KUKA KRL program: ho_lca_st03_pos03.src, ho_lca_st03_pos03.dat

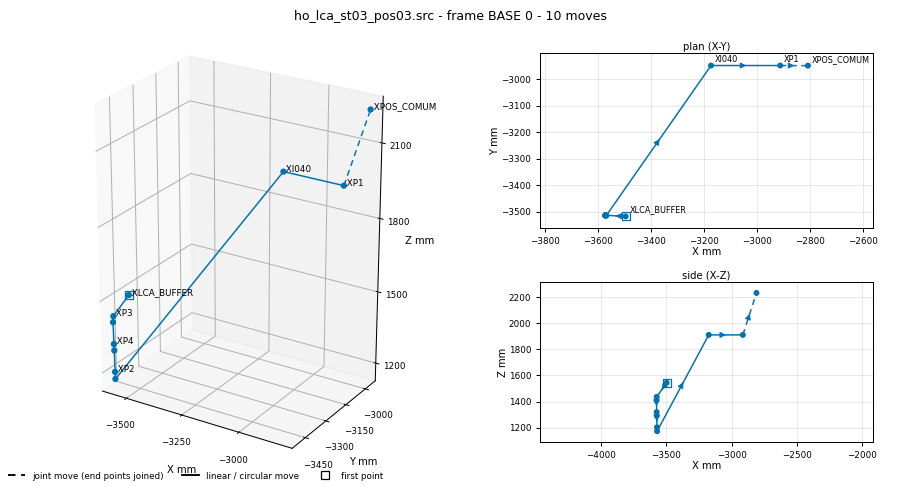
[picture p0: tool path of ho_lca_st03_pos03.src in frame BASE 0, 10 of 10 moves have a stored position in this frame; points joined in program order, loops and branches not executed]
--- ho_lca_st03_pos03.src ---
&ACCESS RVO4
&REL 18
&COMMENT POS_3 LCA
&PARAM DISKPATH = KRC:\R1\Program\LCA
&PARAM TEMPLATE = C:\KRC\Roboter\Template\vorgabe
&PARAM EDITMASK = *
DEF ho_lca_st03_pos03( )
;FOLD INI
  ;FOLD BASISTECH INI
    GLOBAL INTERRUPT DECL 3 WHEN $STOPMESS==TRUE DO IR_STOPM ( )
    INTERRUPT ON 3
    BAS (#INITMOV,0 )
  ;ENDFOLD (BASISTECH INI)
;FOLD GRIPPERTECH INI
USER_GRP(0,DUMMY,DUMMY,GDEFAULT)
;ENDFOLD (GRIPPERTECH INI)
  ;FOLD USER INI
    ;Make your modifications here

  ;ENDFOLD (USER INI)
;ENDFOLD (INI)

; Caracterizacao dos meios de producao:
; Changes: Pega LCA Posicao 3 (Pc-3)
; Versao Atual: 14/08/2015
; Name: P13.050-R2

;FOLD PTP LCA_BUFFER Vel=100 % DEFAULT Tool[15]:AUX_LCA Base[0];%{PE}%R 8.2.20,%MKUKATPBASIS,%CMOVE,%VPTP,%P 1:PTP, 2:LCA_BUFFER, 3:, 5:100, 7:DEFAULT
$BWDSTART=FALSE
PDAT_ACT=PDEFAULT
FDAT_ACT=FLCA_BUFFER
BAS(#PTP_PARAMS,100)
PTP XLCA_BUFFER
;ENDFOLD

;FOLD WAIT FOR ( IN 3362 'LCA p.3' );%{PE}%R 8.2.20,%MKUKATPBASIS,%CEXT_WAIT_FOR,%VEXT_WAIT_FOR,%P 2:, 4:, 5:$IN, 6:3362, 7:LCA p.3, 9:
WAIT FOR  ( $IN[3362] )
;ENDFOLD

;FOLD LIN P3 Vel=1 m/s CPDAT3 Tool[15]:AUX_LCA Base[0];%{PE}%R 8.2.20,%MKUKATPBASIS,%CMOVE,%VLIN,%P 1:LIN, 2:P3, 3:, 5:1, 7:CPDAT3
$BWDSTART=FALSE
LDAT_ACT=LCPDAT3
FDAT_ACT=FP3
BAS(#CP_PARAMS,1)
LIN XP3
;ENDFOLD

;FOLD WAIT FOR ( NOT IN 489 'Presença de peça 1 - Axor LCA' );%{PE}%R 8.2.20,%MKUKATPBASIS,%CEXT_WAIT_FOR,%VEXT_WAIT_FOR,%P 2:, 4:NOT, 5:$IN, 6:489, 7:Presença de peça 1 - Axor LCA, 9:
WAIT FOR  (  NOT $IN[489] )
;ENDFOLD

;FOLD ; POSIÇÃO 1 LCA AUSENTE;%{PE}%R 8.2.20,%MKUKATPBASIS,%CCOMMENT,%VNORMAL,%P 2:POSIÇÃO 1 LCA  AUSENTE
;ENDFOLD
;FOLD LIN PEGA_1 Vel=0.05 m/s L_OLP7 Tool[15]:AUX_LCA Base[0];%{PE}%R 8.2.20,%MKUKATPBASIS,%CMOVE,%VLIN,%P 1:LIN, 2:PEGA_1, 3:, 5:0.05, 7:L_OLP7
$BWDSTART=FALSE
LDAT_ACT=LL_OLP7
FDAT_ACT=FPEGA_1
BAS(#CP_PARAMS,0.05)
LIN XPEGA_1
;ENDFOLD

;FOLD LIN P4 Vel=0.05 m/s CPDAT4 Tool[15]:AUX_LCA Base[0];%{PE}%R 8.2.20,%MKUKATPBASIS,%CMOVE,%VLIN,%P 1:LIN, 2:P4, 3:, 5:0.05, 7:CPDAT4
$BWDSTART=FALSE
LDAT_ACT=LCPDAT4
FDAT_ACT=FP4
BAS(#CP_PARAMS,0.05)
LIN XP4
;ENDFOLD

;FOLD WAIT FOR ( NOT IN 489 'Presença de peça 1 - Axor LCA' );%{PE}%R 8.2.20,%MKUKATPBASIS,%CEXT_WAIT_FOR,%VEXT_WAIT_FOR,%P 2:, 4:NOT, 5:$IN, 6:489, 7:Presença de peça 1 - Axor LCA, 9:
WAIT FOR  (  NOT $IN[489] )
;ENDFOLD

;FOLD ; POSIÇÃO 2 LCA AUSENTE;%{PE}%R 8.2.20,%MKUKATPBASIS,%CCOMMENT,%VNORMAL,%P 2:POSIÇÃO 2 LCA  AUSENTE
;ENDFOLD
;FOLD LIN PEGA_2 Vel=0.05 m/s L_OLP8 Tool[15]:AUX_LCA Base[0];%{PE}%R 8.2.20,%MKUKATPBASIS,%CMOVE,%VLIN,%P 1:LIN, 2:PEGA_2, 3:, 5:0.05, 7:L_OLP8
$BWDSTART=FALSE
LDAT_ACT=LL_OLP8
FDAT_ACT=FPEGA_2
BAS(#CP_PARAMS,0.05)
LIN XPEGA_2
;ENDFOLD

;FOLD LIN P2 Vel=0.05 m/s CPDAT2 Tool[15]:AUX_LCA Base[0];%{PE}%R 8.2.20,%MKUKATPBASIS,%CMOVE,%VLIN,%P 1:LIN, 2:P2, 3:, 5:0.05, 7:CPDAT2
$BWDSTART=FALSE
LDAT_ACT=LCPDAT2
FDAT_ACT=FP2
BAS(#CP_PARAMS,0.05)
LIN XP2
;ENDFOLD

;FOLD ; POSIÇÃO 3 DE PEGA DA PEÇA;%{PE}%R 8.2.20,%MKUKATPBASIS,%CCOMMENT,%VNORMAL,%P 2:POSIÇÃO  3 DE PEGA DA PEÇA
;ENDFOLD
;FOLD LIN PEGA_3 Vel=0.05 m/s L_OLP5 Tool[15]:AUX_LCA Base[0];%{PE}%R 8.2.20,%MKUKATPBASIS,%CMOVE,%VLIN,%P 1:LIN, 2:PEGA_3, 3:, 5:0.05, 7:L_OLP5
$BWDSTART=FALSE
LDAT_ACT=LL_OLP5
FDAT_ACT=FPEGA_3
BAS(#CP_PARAMS,0.05)
LIN XPEGA_3
;ENDFOLD

IF (NOT(GHOST())) THEN
;FOLD WAIT FOR ( IN 489 'Presença de peça 1 - Axor' );%{PE}%R 8.2.20,%MKUKATPBASIS,%CEXT_WAIT_FOR,%VEXT_WAIT_FOR,%P 2:, 4:, 5:$IN, 6:489, 7:Presença de peça 1 - Axor, 9:
WAIT FOR  ( $IN[489] )
;ENDFOLD
ENDIF

;FOLD SET Z4.1 GRP AXOR State=CLO GDAT6;%{PE}%R 8.2.1,%MKUKATPGRP,%CGRP,%VGRP,%P 2:12, 4:2, 5:#NO, 6:GDAT6, 8:0, 10:0
H50(GRP,12,2,GGDAT6)
;ENDFOLD
chk_w6_grp4_clo()

IF (NOT(GHOST())) THEN
;FOLD SET VACUO AXOR State=VACUUM GDAT7;%{PE}%R 8.2.1,%MKUKATPGRP,%CGRP,%VGRP,%P 2:9, 4:1, 5:#NO, 6:GDAT7, 8:0, 10:0
H50(GRP,9,1,GGDAT7)
;ENDFOLD
chk_w6_grp1_vac()
ENDIF

;FOLD OUT 3371 'Lib. p/ sair c/ Travessa Axor/Atego' State=TRUE ;%{PE}%R 8.2.20,%MKUKATPBASIS,%COUT,%VOUTX,%P 2:3371, 3:Lib. p/ sair c/ Travessa Axor/Atego, 5:TRUE, 6:
$OUT[3371]=TRUE
;ENDFOLD
;FOLD WAIT Time=1 sec;%{PE}%R 8.2.20,%MKUKATPBASIS,%CWAIT,%VWAIT,%P 3:1
WAIT SEC 1
;ENDFOLD
;FOLD WAIT FOR ( IN 3371 'Lib. p/ Sair c/ Pç LCA Axor/Atego' );%{PE}%R 8.2.20,%MKUKATPBASIS,%CEXT_WAIT_FOR,%VEXT_WAIT_FOR,%P 2:, 4:, 5:$IN, 6:3371, 7:Lib. p/ Sair c/ Pç LCA Axor/Atego, 9:
WAIT FOR  ( $IN[3371] )
;ENDFOLD
;FOLD OUT 3371 'Lib. p/ sair c/ Travessa Axor/Atego' State=FALSE ;%{PE}%R 8.2.20,%MKUKATPBASIS,%COUT,%VOUTX,%P 2:3371, 3:Lib. p/ sair c/ Travessa Axor/Atego, 5:FALSE, 6:
$OUT[3371]=FALSE
;ENDFOLD
;FOLD OUT 3349 'R2 pegou peça' State=FALSE ;%{PE}%R 8.2.20,%MKUKATPBASIS,%COUT,%VOUTX,%P 2:3349, 3:R2 pegou peça, 5:FALSE, 6:
$OUT[3349]=FALSE
;ENDFOLD

;FOLD LIN l040 Vel=0.02 m/s L_OLP6 Tool[6]:Gripper G0100R Base[0];%{PE}%R 8.2.20,%MKUKATPBASIS,%CMOVE,%VLIN,%P 1:LIN, 2:l040, 3:, 5:0.02, 7:L_OLP6
$BWDSTART=FALSE
LDAT_ACT=LL_OLP6
FDAT_ACT=Fl040
BAS(#CP_PARAMS,0.02)
LIN Xl040
;ENDFOLD

;FOLD WAIT FOR ( IN 489 'Presença de peça 1 - Axor LCA' OR Ghost() );%{PE}%R 8.2.20,%MKUKATPBASIS,%CEXT_WAIT_FOR,%VEXT_WAIT_FOR,%P 2:, 4:, 5:$IN, 6:489, 7:Presença de peça 1 - Axor LCA, 8:OR, 9:, 10:Ghost(), 11:489, 12:, 14:
WAIT FOR  ( $IN[489] OR Ghost() )
;ENDFOLD

;FOLD LIN P1 Vel=0.05 m/s CPDAT1 Tool[6]:Gripper G0100R Base[0];%{PE}%R 8.2.20,%MKUKATPBASIS,%CMOVE,%VLIN,%P 1:LIN, 2:P1, 3:, 5:0.05, 7:CPDAT1
$BWDSTART=FALSE
LDAT_ACT=LCPDAT1
FDAT_ACT=FP1
BAS(#CP_PARAMS,0.05)
LIN XP1
;ENDFOLD

;FOLD ; POSIÇÃO COMUM;%{PE}%R 8.2.20,%MKUKATPBASIS,%CCOMMENT,%VNORMAL,%P 2:POSIÇÃO COMUM
;ENDFOLD
;FOLD PTP POS_COMUM Vel=100 % PDAT0 Tool[6]:Gripper G0100R Base[0];%{PE}%R 8.2.20,%MKUKATPBASIS,%CMOVE,%VPTP,%P 1:PTP, 2:POS_COMUM, 3:, 5:100, 7:PDAT0
$BWDSTART=FALSE
PDAT_ACT=PPDAT0
FDAT_ACT=FPOS_COMUM
BAS(#PTP_PARAMS,100)
PTP XPOS_COMUM
;ENDFOLD

END

--- ho_lca_st03_pos03.dat ---
&ACCESS RVO4
&REL 18
&COMMENT POS_3 LCA
&PARAM DISKPATH = KRC:\R1\Program\LCA
&PARAM TEMPLATE = C:\KRC\Roboter\Template\vorgabe
&PARAM EDITMASK = *
DEFDAT  ho_lca_st03_pos03
;FOLD EXTERNAL DECLARATIONS;%{PE}%MKUKATPBASIS,%CEXT,%VCOMMON,%P
;FOLD GRIPPERTECH EXT
EXT  H50 (INT  :IN,INT  :IN,INT  :IN,GRP_TYP  :IN )
;ENDFOLD (GRIPPERTECH EXT)
;FOLD SPOTTECH EXT
EXT  USERSPOT (S_COMMAND  :IN,SPOT_TYPE  :IN )
;ENDFOLD (SPOTTECH EXT)
;FOLD BASISTECH EXT;%{PE}%MKUKATPBASIS,%CEXT,%VEXT,%P
EXT  BAS (BAS_COMMAND  :IN,REAL  :IN )
DECL INT SUCCESS
;ENDFOLD (BASISTECH EXT)
;FOLD USER EXT;%{E}%MKUKATPUSER,%CEXT,%VEXT,%P
;Make your modifications here

;ENDFOLD (USER EXT)
;ENDFOLD (EXTERNAL DECLARATIONS)
DECL BASIS_SUGG_T LAST_BASIS={POINT1[] "P4                      ",POINT2[] "P4                      ",CP_PARAMS[] "CPDAT4                  ",PTP_PARAMS[] "PDAT0                   ",CONT[] "                        ",CP_VEL[] "0.05                    ",PTP_VEL[] "100                     ",SYNC_PARAMS[] "SYNCDAT                 ",SPL_NAME[] "S0                      "}
DECL LDAT LL_OLP5={VEL 0.25,ACC 100.0,APO_DIST 0.0,APO_FAC 0.0,ORI_TYP #VAR,CIRC_TYP #BASE,JERK_FAC 50.0}
DECL GRP_SUGG_T LAST_GRP={NUMBER[] "9                       ",STATE[] "1                       ",PARAMS[] "GDAT1                   "}
DECL GRP_TYP GGDAT6={G_APO #NO,GRP_TIME 0.200000003,CTRL #OFF,DLY 0,DST 1}
DECL LDAT LL_OLP6={VEL 0.25,ACC 100.0,APO_DIST 0.0,APO_FAC 0.0,ORI_TYP #VAR,CIRC_TYP #BASE,JERK_FAC 50.0}
DECL E6POS Xl040={X -3174.60205,Y -2948.20093,Z 1910.30298,A -158.906006,B 84.1113815,C 96.0123901,S 2,T 34,E1 3299.98706,E2 0.0,E3 0.0,E4 0.0,E5 0.0,E6 0.0}
DECL FDAT Fl040={TOOL_NO 6,BASE_NO 0,IPO_FRAME #BASE,POINT2[] " ",TQ_STATE FALSE}
DECL GRP_TYP GGDAT1={G_APO #NO,GRP_TIME 0.200000003,CTRL #OFF,DLY 0,DST 1}
DECL GRP_TYP GGDAT2={G_APO #NO,GRP_TIME 0.200000003,CTRL #OFF,DLY 0,DST 1}
DECL PDAT PPDAT0={VEL 100.0,ACC 100.0,APO_DIST 100.0}
DECL E6POS XPOS_COMUM={X -2809.396,Y -2948.65088,Z 2231.30811,A -163.868805,B 82.3905334,C 90.4837494,S 2,T 34,E1 3299.98706,E2 0.0,E3 0.0,E4 0.0,E5 0.0,E6 0.0}
DECL FDAT FPOS_COMUM={TOOL_NO 6,BASE_NO 0,IPO_FRAME #BASE,POINT2[] " ",TQ_STATE FALSE}
DECL GRP_TYP GGDAT3={G_APO #NO,GRP_TIME 0.200000003,CTRL #OFF,DLY 0,DST 1}
DECL GRP_TYP GGDAT4={G_APO #NO,GRP_TIME 0.200000003,CTRL #OFF,DLY 0,DST 1}
DECL E6POS XP1={X -2913.604,Y -2948.19995,Z 1910.297,A -158.903305,B 84.1116409,C 96.0151291,S 2,T 34,E1 3299.98706,E2 0.0,E3 0.0,E4 0.0,E5 0.0,E6 0.0}
DECL FDAT FP1={TOOL_NO 6,BASE_NO 0,IPO_FRAME #BASE,POINT2[] " ",TQ_STATE FALSE}
DECL LDAT LCPDAT1={VEL 2.0,ACC 100.0,APO_DIST 100.0,APO_FAC 50.0,AXIS_VEL 100.0,AXIS_ACC 100.0,ORI_TYP #VAR,CIRC_TYP #BASE,JERK_FAC 50.0,GEAR_JERK 50.0,EXAX_IGN 0}
DECL GRP_TYP GGDAT5={G_APO #NO,GRP_TIME 0.200000003,CTRL #OFF,DLY 0,DST 1}
DECL GRP_TYP GGDAT7={G_APO #NO,GRP_TIME 0.200000003,CTRL #OFF,DLY 0,DST 1}
DECL E6POS XLCA_BUFFER={X -3496.6189,Y -3516.89502,Z 1544.35803,A -172.404495,B -1.92999804,C -179.6474,S 2,T 34,E1 3299.98901,E2 0.0,E3 0.0,E4 0.0,E5 0.0,E6 0.0}
DECL FDAT FLCA_BUFFER={TOOL_NO 15,BASE_NO 0,IPO_FRAME #BASE,POINT2[] " ",TQ_STATE FALSE}
DECL E6POS XP2={X -3570.20801,Y -3514.07397,Z 1203.78003,A -172.936798,B -0.115350299,C 179.957001,S 2,T 34,E1 3299.98511,E2 0.0,E3 0.0,E4 0.0,E5 0.0,E6 0.0}
DECL FDAT FP2={TOOL_NO 15,BASE_NO 0,IPO_FRAME #BASE,POINT2[] " ",TQ_STATE FALSE}
DECL LDAT LCPDAT2={VEL 2.0,ACC 100.0,APO_DIST 100.0,APO_FAC 50.0,AXIS_VEL 100.0,AXIS_ACC 100.0,ORI_TYP #VAR,CIRC_TYP #BASE,JERK_FAC 50.0,GEAR_JERK 50.0,EXAX_IGN 0}
DECL E6POS XPEGA_5={X -3571.42798,Y -3513.94092,Z 1173.70496,A -172.937195,B -0.118930399,C 179.957993,S 2,T 34,E1 3299.98804,E2 0.0,E3 0.0,E4 0.0,E5 0.0,E6 0.0}
DECL FDAT FPEGA_5={TOOL_NO 15,BASE_NO 0,IPO_FRAME #BASE,POINT2[] " ",TQ_STATE FALSE}
DECL E6POS XPEGA_3={X -3569.61597,Y -3513.95288,Z 1173.68896,A -172.937103,B -0.118397102,C 179.957794,S 2,T 34,E1 3299.98608,E2 0.0,E3 0.0,E4 0.0,E5 0.0,E6 0.0}
DECL FDAT FPEGA_3={TOOL_NO 15,BASE_NO 0,IPO_FRAME #BASE,POINT2[] " ",TQ_STATE FALSE}
DECL LDAT LCPDAT3={VEL 2.0,ACC 100.0,APO_DIST 100.0,APO_FAC 50.0,AXIS_VEL 100.0,AXIS_ACC 100.0,ORI_TYP #VAR,CIRC_TYP #BASE,JERK_FAC 50.0,GEAR_JERK 50.0,EXAX_IGN 0}
DECL E6POS XP3={X -3572.30103,Y -3512.85303,Z 1436.37097,A -172.186798,B -1.49960494,C -179.705902,S 2,T 34,E1 3299.97998,E2 0.0,E3 0.0,E4 0.0,E5 0.0,E6 0.0}
DECL FDAT FP3={TOOL_NO 15,BASE_NO 0,IPO_FRAME #BASE,POINT2[] " ",TQ_STATE FALSE}
DECL LDAT LL_OLP7={VEL 0.25,ACC 100.0,APO_DIST 0.0,APO_FAC 0.0,ORI_TYP #VAR,CIRC_TYP #BASE,JERK_FAC 50.0}
DECL E6POS XPEGA_1={X -3573.979,Y -3513.69092,Z 1411.08704,A -172.191803,B -1.54883206,C -179.901199,S 2,T 34,E1 3299.979,E2 0.0,E3 0.0,E4 0.0,E5 0.0,E6 0.0}
DECL FDAT FPEGA_1={TOOL_NO 15,BASE_NO 0,IPO_FRAME #BASE,POINT2[] " ",TQ_STATE FALSE}
DECL LDAT LCPDAT4={VEL 2.0,ACC 100.0,APO_DIST 100.0,APO_FAC 50.0,AXIS_VEL 100.0,AXIS_ACC 100.0,ORI_TYP #VAR,CIRC_TYP #BASE,JERK_FAC 50.0,GEAR_JERK 50.0,EXAX_IGN 0}
DECL E6POS XP4={X -3573.13306,Y -3512.88501,Z 1319.96997,A -172.473206,B -0.122878,C -179.874893,S 2,T 34,E1 3299.98706,E2 0.0,E3 0.0,E4 0.0,E5 0.0,E6 0.0}
DECL FDAT FP4={TOOL_NO 15,BASE_NO 0,IPO_FRAME #BASE,POINT2[] " ",TQ_STATE FALSE}
DECL LDAT LL_OLP8={VEL 0.25,ACC 100.0,APO_DIST 0.0,APO_FAC 0.0,ORI_TYP #VAR,CIRC_TYP #BASE,JERK_FAC 50.0}
DECL E6POS XPEGA_2={X -3572.448,Y -3512.36108,Z 1292.95996,A -172.473099,B -0.122928903,C -179.875198,S 2,T 34,E1 3299.98706,E2 0.0,E3 0.0,E4 0.0,E5 0.0,E6 0.0}
DECL FDAT FPEGA_2={TOOL_NO 15,BASE_NO 0,IPO_FRAME #BASE,POINT2[] " ",TQ_STATE FALSE}
ENDDAT
